PROGRAM Axis01_Command
VAR
//System_Bit
	Always_ON	:	BOOL	:=TRUE	;//상시 ON 
	Always_OFF	:	BOOL	:=FALSE	;//상시 OFF	

//Motor
	Axis01_MC_Power: MC_Power;
	Axis01: AXIS_REF;										//Guide축
	Axis01_MC_Home: FB_HomeBeforeMoveAX8000;
	Axis01_Jog: MC_Jog;
	Axis01_Home_Pos_Move: MC_MoveAbsolute;						//Home 방향 변경불가 Home 동작 전 Sensor앞 으로 이동
	Axis01_Wait_Pos_Move: MC_MoveAbsolute;
	Axis01_Target_Pos_Move: MC_MoveAbsolute;
	Axis01_Work_End_Pos_Move: MC_MoveAbsolute;
	Axis01_Maint_Pos_Move: MC_MoveAbsolute;
	Axis01_Tool_Change_Pos_Move: MC_MoveAbsolute;
	Axis01_Calibration_Pos_Move: MC_MoveAbsolute;
	Axis01_Product_Pos_Move: MC_MoveAbsolute;
END_VAR
VAR // added by the converter: edge detectors and wires of the graphical bodies
    _rt1 : R_TRIG;
END_VAR

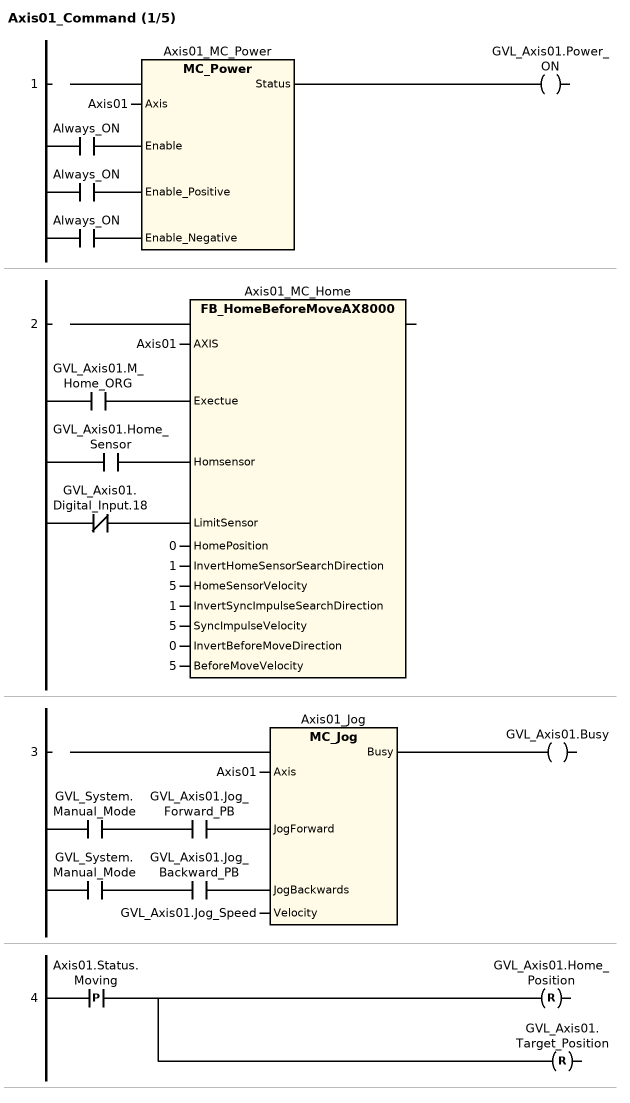
// NETWORK 1
Axis01_MC_Power(
    Axis := Axis01,
    Enable := Always_ON,
    Enable_Positive := Always_ON,
    Enable_Negative := Always_ON); // MC_Power
GVL_Axis01.Power_ON := Axis01_MC_Power.Status;

// NETWORK 2
Axis01_MC_Home(
    AXIS := Axis01,
    Exectue := GVL_Axis01.M_Home_ORG,
    Homsensor := GVL_Axis01.Home_Sensor,
    LimitSensor := NOT GVL_Axis01.Digital_Input.18,
    HomePosition := 0,
    InvertHomeSensorSearchDirection := 1,
    HomeSensorVelocity := 5,
    InvertSyncImpulseSearchDirection := 1,
    SyncImpulseVelocity := 5,
    InvertBeforeMoveDirection := 0,
    BeforeMoveVelocity := 5); // FB_HomeBeforeMoveAX8000

// NETWORK 3
Axis01_Jog(
    Axis := Axis01,
    JogForward := GVL_System.Manual_Mode AND GVL_Axis01.Jog_Forward_PB,
    JogBackwards := GVL_System.Manual_Mode AND GVL_Axis01.Jog_Backward_PB,
    Velocity := GVL_Axis01.Jog_Speed,
    Busy => GVL_Axis01.Busy); // MC_Jog

// NETWORK 4
_rt1(CLK := Axis01.Status.Moving);
GVL_Axis01.Home_Position R= _rt1.Q;
GVL_Axis01.Target_Position R= _rt1.Q;

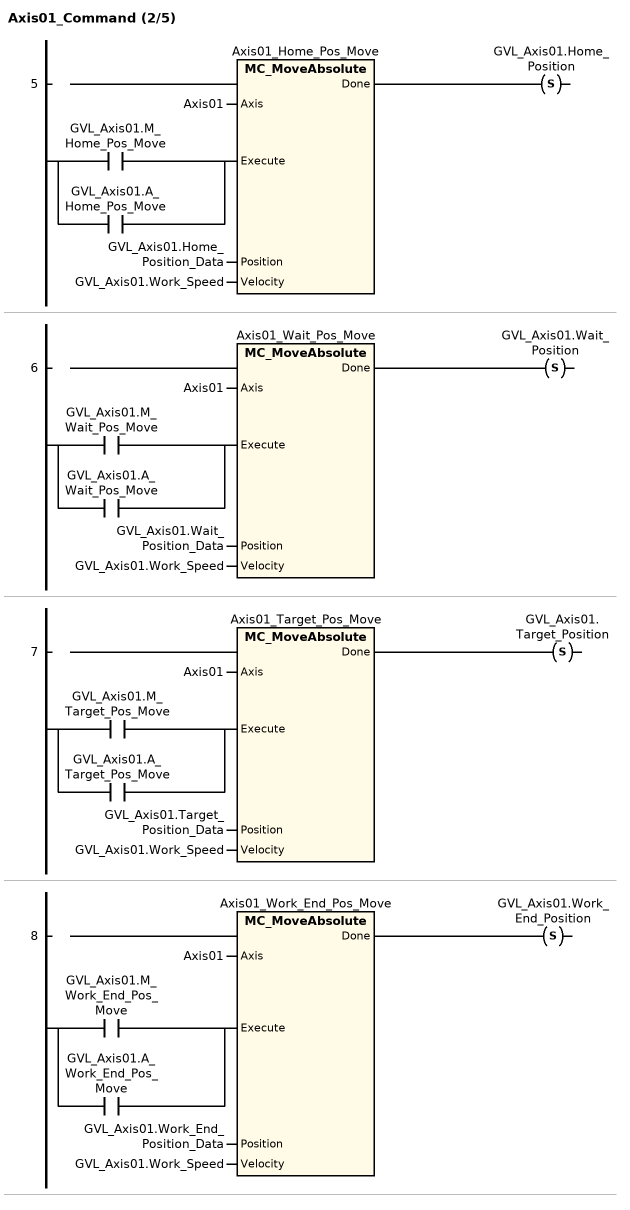
// NETWORK 5
Axis01_Home_Pos_Move(
    Axis := Axis01,
    Execute := GVL_Axis01.M_Home_Pos_Move OR GVL_Axis01.A_Home_Pos_Move,
    Position := GVL_Axis01.Home_Position_Data,
    Velocity := GVL_Axis01.Work_Speed); // MC_MoveAbsolute
GVL_Axis01.Home_Position S= Axis01_Home_Pos_Move.Done;

// NETWORK 6
Axis01_Wait_Pos_Move(
    Axis := Axis01,
    Execute := GVL_Axis01.M_Wait_Pos_Move OR GVL_Axis01.A_Wait_Pos_Move,
    Position := GVL_Axis01.Wait_Position_Data,
    Velocity := GVL_Axis01.Work_Speed); // MC_MoveAbsolute
GVL_Axis01.Wait_Position S= Axis01_Wait_Pos_Move.Done;

// NETWORK 7
Axis01_Target_Pos_Move(
    Axis := Axis01,
    Execute := GVL_Axis01.M_Target_Pos_Move OR GVL_Axis01.A_Target_Pos_Move,
    Position := GVL_Axis01.Target_Position_Data,
    Velocity := GVL_Axis01.Work_Speed); // MC_MoveAbsolute
GVL_Axis01.Target_Position S= Axis01_Target_Pos_Move.Done;

// NETWORK 8
Axis01_Work_End_Pos_Move(
    Axis := Axis01,
    Execute := GVL_Axis01.M_Work_End_Pos_Move OR GVL_Axis01.A_Work_End_Pos_Move,
    Position := GVL_Axis01.Work_End_Position_Data,
    Velocity := GVL_Axis01.Work_Speed); // MC_MoveAbsolute
GVL_Axis01.Work_End_Position S= Axis01_Work_End_Pos_Move.Done;

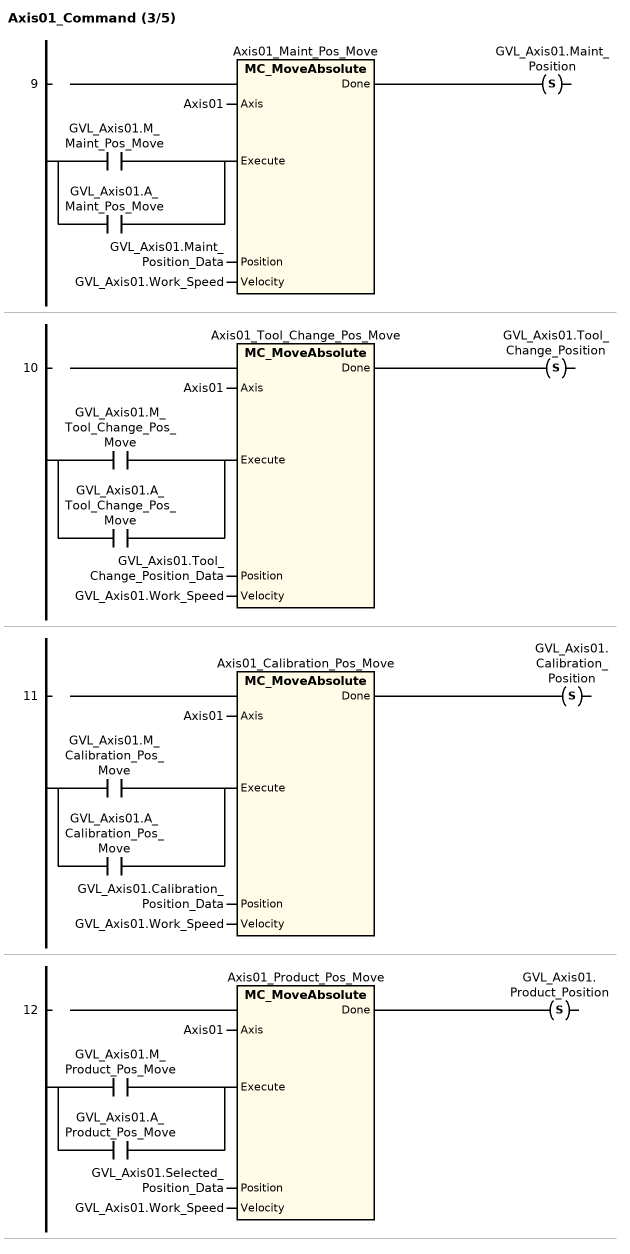
// NETWORK 9
Axis01_Maint_Pos_Move(
    Axis := Axis01,
    Execute := GVL_Axis01.M_Maint_Pos_Move OR GVL_Axis01.A_Maint_Pos_Move,
    Position := GVL_Axis01.Maint_Position_Data,
    Velocity := GVL_Axis01.Work_Speed); // MC_MoveAbsolute
GVL_Axis01.Maint_Position S= Axis01_Maint_Pos_Move.Done;

// NETWORK 10
Axis01_Tool_Change_Pos_Move(
    Axis := Axis01,
    Execute := GVL_Axis01.M_Tool_Change_Pos_Move OR GVL_Axis01.A_Tool_Change_Pos_Move,
    Position := GVL_Axis01.Tool_Change_Position_Data,
    Velocity := GVL_Axis01.Work_Speed); // MC_MoveAbsolute
GVL_Axis01.Tool_Change_Position S= Axis01_Tool_Change_Pos_Move.Done;

// NETWORK 11
Axis01_Calibration_Pos_Move(
    Axis := Axis01,
    Execute := GVL_Axis01.M_Calibration_Pos_Move OR GVL_Axis01.A_Calibration_Pos_Move,
    Position := GVL_Axis01.Calibration_Position_Data,
    Velocity := GVL_Axis01.Work_Speed); // MC_MoveAbsolute
GVL_Axis01.Calibration_Position S= Axis01_Calibration_Pos_Move.Done;

// NETWORK 12
Axis01_Product_Pos_Move(
    Axis := Axis01,
    Execute := GVL_Axis01.M_Product_Pos_Move OR GVL_Axis01.A_Product_Pos_Move,
    Position := GVL_Axis01.Selected_Position_Data,
    Velocity := GVL_Axis01.Work_Speed); // MC_MoveAbsolute
GVL_Axis01.Product_Position S= Axis01_Product_Pos_Move.Done;

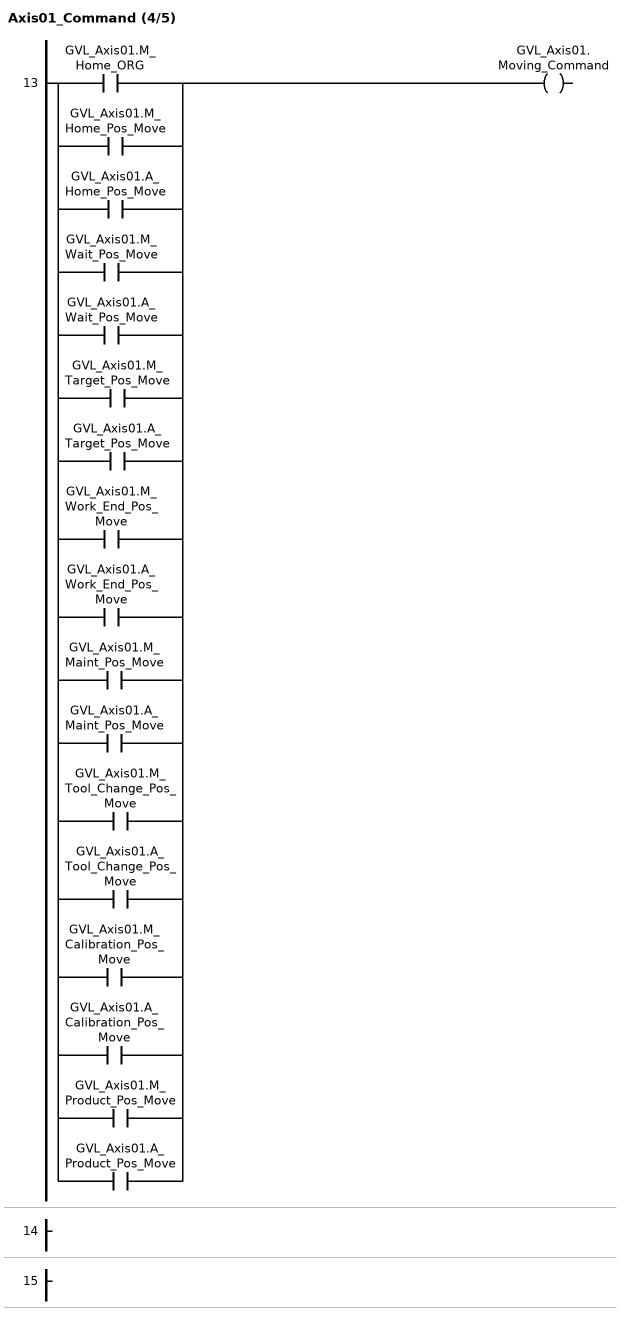
// NETWORK 13
GVL_Axis01.Moving_Command := GVL_Axis01.M_Home_ORG OR GVL_Axis01.M_Home_Pos_Move OR GVL_Axis01.A_Home_Pos_Move OR GVL_Axis01.M_Wait_Pos_Move OR GVL_Axis01.A_Wait_Pos_Move OR GVL_Axis01.M_Target_Pos_Move OR GVL_Axis01.A_Target_Pos_Move OR GVL_Axis01.M_Work_End_Pos_Move OR GVL_Axis01.A_Work_End_Pos_Move OR GVL_Axis01.M_Maint_Pos_Move OR GVL_Axis01.A_Maint_Pos_Move OR GVL_Axis01.M_Tool_Change_Pos_Move OR GVL_Axis01.A_Tool_Change_Pos_Move OR GVL_Axis01.M_Calibration_Pos_Move OR GVL_Axis01.A_Calibration_Pos_Move OR GVL_Axis01.M_Product_Pos_Move OR GVL_Axis01.A_Product_Pos_Move;

// NETWORK 14

// NETWORK 15

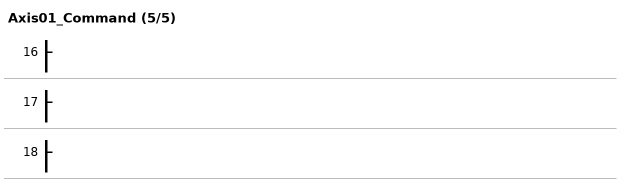
// NETWORK 16

// NETWORK 17

// NETWORK 18

END_PROGRAM

(* stored: Version 1.1.0.1, ProductVersion 3.1.4024.15
   POU Axis01_Command: Id {b0aad668-381a-4d39-86df-d8cdc6cf7674}, SpecialFunc None *)
